Universal Robots PolyScope program: bearing_plate_pick.urp

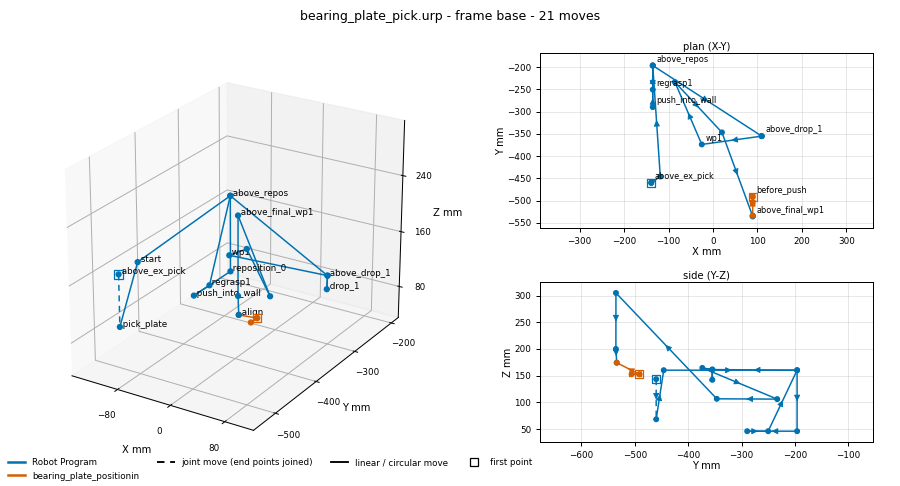
[picture p0: tool path of bearing_plate_pick.urp in frame base, 21 of 22 moves have a stored position in this frame; points joined in program order, loops and branches not executed]
Program bearing_plate_pick (installation=default directory=/programs/wrs2020 createdIn=5.6.0.90886 lastSavedIn=5.9.1.1031110 robotSerialNumber=20205500180)
Calibrated DH parameters: a=[0, -0.425, -0.3922, 0, 0, 0]; d=[0.1625, 0, 0, 0.1333, 0.0997, 0.0996]; alpha=[1.570796, 0, 0, 1.570796, -1.570796, 0]; deltaTheta=[0, 0, 0, 0, 0, 0]
Robot Program (runOnlyOnce=true)
  MoveJ speed 60 deg/s, acceleration 80 deg/s^2 (useActiveTCP=true) feature=Base
    currentpose := get_actual_tcp_pose()get_actual_joint_positions()
    Waypoint Waypoint (Variable): variable=currentpose
  MoveJ speed 60 deg/s, acceleration 80 deg/s^2 (useActiveTCP=true) feature=Base
    URCap Gripper (Robotiq_Grippers, Robotiq Inc.) dataModel(position=64.70588235294117, force=0.0, speed=0.0, positionInDouble=64.70588235294117, forceInDouble=0.0, speedInDouble=0.0, slaveIds=[9], blocking=true)
    Waypoint above_ex_pick: TCP in base x=-139.039 y=-460.061 z=143.501 mm, rx=-2.2048 ry=-2.2054 rz=0.0296 rad; joints [58.139, -91.524, 110.219, -109.456, -91.532, 58.113] deg; TCP offset x=0 y=0 z=220 mm, rx=0 ry=0 rz=0 rad
    Waypoint pick_plate: TCP in base x=-139.031 y=-460.052 z=68.363 mm, rx=-2.2048 ry=-2.2054 rz=0.0296 rad; joints [58.14, -86.891, 117.616, -121.485, -91.533, 58.114] deg; TCP offset x=0 y=0 z=220 mm, rx=0 ry=0 rz=0 rad
    URCap Gripper (Robotiq_Grippers, Robotiq Inc.) dataModel(position=100.0, force=0.0, speed=0.0, positionInDouble=100.0, forceInDouble=0.0, speedInDouble=0.0, slaveIds=[9], blocking=true)
  Folder Rearrange
    MoveL speed 800 mm/s, acceleration 1200 mm/s^2 (useActiveTCP=false) tcp=gripper_140_tip; feature=Base
      Waypoint start: motionParameters(blendRadius=0.03); TCP in base x=-118.669 y=-445.946 z=160.266 mm, rx=2.1923 ry=2.2501 rz=0.0089 rad; joints [58.256, -94.58, 110.219, -105.321, -89.927, 56.766] deg; TCP offset x=0 y=0 z=220 mm, rx=0 ry=0 rz=0 rad
      Waypoint above_repos: motionParameters(blendRadius=0.05); TCP in base x=-135.607 y=-196.202 z=160.258 mm, rx=3.137 ry=-0.0475 rz=0.0061 rad; joints [20.876, -133.857, 132.235, -88.26, -89.695, 112.61] deg; TCP offset x=0 y=0 z=220 mm, rx=0 ry=0 rz=0 rad
      Waypoint reposition_0: TCP in base x=-135.6 y=-196.2 z=46.036 mm, rx=3.1371 ry=-0.0475 rz=0.0061 rad; joints [20.876, -130.464, 148.282, -107.699, -89.695, 112.611] deg
      URCap Gripper (Robotiq_Grippers, Robotiq Inc.) dataModel(position=72.54901960784314, force=0.0, speed=0.0, positionInDouble=72.54901960784314, forceInDouble=0.0, speedInDouble=0.0, slaveIds=[9], blocking=true)
      URCap Gripper (Robotiq_Grippers, Robotiq Inc.) dataModel(position=83.92156862745098, force=0.0, speed=0.0, positionInDouble=83.92156862745098, forceInDouble=0.0, speedInDouble=0.0, slaveIds=[9], blocking=true)
      Waypoint push_into_wall: TCP in base x=-135.617 y=-289.652 z=46.047 mm, rx=3.137 ry=-0.0475 rz=0.0061 rad; joints [39.919, -110.73, 140.431, -119.691, -89.673, 131.655] deg
      URCap Gripper (Robotiq_Grippers, Robotiq Inc.) dataModel(position=72.54901960784314, force=0.0, speed=0.0, positionInDouble=72.54901960784314, forceInDouble=0.0, speedInDouble=0.0, slaveIds=[9], blocking=true)
      Waypoint regrasp1: TCP in base x=-135.589 y=-250.402 z=46.038 mm, rx=3.1371 ry=-0.0475 rz=0.0061 rad; joints [33.242, -118.348, 144.167, -115.768, -89.677, 124.976] deg
      URCap Gripper (Robotiq_Grippers, Robotiq Inc.) dataModel(position=100.0, force=0.0, speed=0.0, positionInDouble=100.0, forceInDouble=0.0, speedInDouble=0.0, slaveIds=[9], blocking=true)
      Waypoint above_repos: TCP in base x=-135.607 y=-196.202 z=160.258 mm, rx=3.137 ry=-0.0475 rz=0.0061 rad; joints [20.876, -133.857, 132.235, -88.26, -89.695, 112.61] deg
      URCap Gripper (Robotiq_Grippers, Robotiq Inc.) dataModel(position=100.0, force=0.0, speed=0.0, positionInDouble=100.0, forceInDouble=0.0, speedInDouble=0.0, slaveIds=[9], blocking=true)
  MoveL speed 800 mm/s, acceleration 1200 mm/s^2 (useActiveTCP=false) tcp=gripper_140_tip; feature=Base
    SuppressedNode
      Waypoint start: TCP in base x=-118.669 y=-445.946 z=160.266 mm, rx=2.1923 ry=2.2501 rz=0.0089 rad; joints [58.256, -94.58, 110.219, -105.321, -89.927, 56.766] deg; TCP offset x=0 y=0 z=220 mm, rx=0 ry=0 rz=0 rad
    Waypoint above_drop_1: TCP in base x=109.642 y=-355.035 z=161.42 mm, rx=0.0416 ry=-3.1373 rz=-0.0063 rad; joints [86.366, -108.401, 120.826, -102.213, -90.247, -5.154] deg; TCP offset x=0 y=0 z=220 mm, rx=0 ry=0 rz=0 rad
    Waypoint drop_1: TCP in base x=109 y=-355.041 z=142.278 mm, rx=0.0417 ry=-3.1373 rz=-0.0063 rad; joints [86.261, -107.694, 123.246, -105.338, -90.248, -5.26] deg; TCP offset x=0 y=0 z=220 mm, rx=0 ry=0 rz=0 rad
    URCap Gripper (Robotiq_Grippers, Robotiq Inc.) dataModel(position=72.54901960784314, force=0.0, speed=0.0, positionInDouble=72.54901960784314, forceInDouble=0.0, speedInDouble=0.0, slaveIds=[9], blocking=true)
    Waypoint above_drop_1: TCP in base x=109.642 y=-355.035 z=161.42 mm, rx=0.0416 ry=-3.1373 rz=-0.0063 rad; joints [86.366, -108.401, 120.826, -102.213, -90.247, -5.154] deg; TCP offset x=0 y=0 z=220 mm, rx=0 ry=0 rz=0 rad
    Waypoint wp1: motionParameters(blendRadius=0.05); TCP in base x=-25.271 y=-373.698 z=164.531 mm, rx=0.4375 ry=2.7113 rz=-0.1186 rad; joints [44.743, -110.618, 123.094, -92.727, -69.038, -28.731] deg; TCP offset x=0 y=0 z=220 mm, rx=0 ry=0 rz=0 rad
    Waypoint before_grasp: motionParameters(jointSpeed=1.047198 jointAcceleration=1.396263 cartesianSpeed=0.25 cartesianAcceleration=1.2 blendRadius=0.02); TCP in base x=-85.778 y=-233.44 z=106.112 mm, rx=0.6196 ry=1.477 rz=-0.6265 rad; joints [-24.668, -72.215, 139.816, -67.364, -68.98, -90.257] deg
    Waypoint at_grasp: motionParameters(jointSpeed=1.047198 jointAcceleration=1.396263 cartesianSpeed=0.25 cartesianAcceleration=1.2); TCP in base x=20.032 y=-346.58 z=106.691 mm, rx=0.6197 ry=1.477 rz=-0.6265 rad; joints [-4.452, -79.298, 152.241, -72.65, -48.761, -90.363] deg
    URCap Gripper (Robotiq_Grippers, Robotiq Inc.) dataModel(position=100.0, force=0.0, speed=0.0, positionInDouble=100.0, forceInDouble=0.0, speedInDouble=0.0, slaveIds=[9], blocking=true)
    MoveDirectionNode (toolParams=0.8, 0.4) expression=[-0.3,0.0,1.0]
      Until DISTANCE (allowActions=false deceleration=3 distanceNodeType=BLEND) Distance=0.15; motionParameters(blendRadius=0.08)
    Waypoint above_final_wp1: motionParameters(jointSpeed=1.047198 jointAcceleration=1.396263 cartesianSpeed=0.8 cartesianAcceleration=0.4 blendRadius=0.03); TCP in base x=89.208 y=-535.392 z=304.9 mm, rx=0.0022 ry=-2.7904 rz=1.4282 rad; joints [80.944, -112.949, 134.272, -165.222, -82.979, -5.575] deg
    Waypoint place: motionParameters(jointSpeed=1.047198 jointAcceleration=1.396263 cartesianSpeed=0.8 cartesianAcceleration=0.4); TCP in base x=89.218 y=-535.49 z=200.099 mm, rx=0.0021 ry=-2.8448 rz=1.3158 rad; joints [81.498, -103.024, 141.717, -178.058, -83.875, -5.768] deg
    URCap Gripper (Robotiq_Grippers, Robotiq Inc.) dataModel(position=72.54901960784314, force=0.0, speed=0.0, positionInDouble=72.54901960784314, forceInDouble=0.0, speedInDouble=0.0, slaveIds=[9], blocking=true)
    Waypoint align: TCP in base x=89.24 y=-533.942 z=174.306 mm, rx=0.0138 ry=2.8434 rz=-1.3083 rad; joints [80.63, -99.836, 144.208, -183.367, -82.506, -5.396] deg
    URCap Gripper (Robotiq_Grippers, Robotiq Inc.) dataModel(position=100.0, force=0.0, speed=0.0, positionInDouble=100.0, forceInDouble=0.0, speedInDouble=0.0, slaveIds=[9], blocking=true)
    URCap Gripper (Robotiq_Grippers, Robotiq Inc.) dataModel(position=72.54901960784314, force=0.0, speed=0.0, positionInDouble=72.54901960784314, forceInDouble=0.0, speedInDouble=0.0, slaveIds=[9], blocking=true)
  Call bearing_plate_positioning
SubProgram -> bearing_plate_positioning
SubProgram bearing_plate_positioning (keepSynchronizedWithDisk=true) programFile=/programs/wrs2020/bearing_plate_positioning.urp
  MoveL speed 250 mm/s, acceleration 1200 mm/s^2 (useActiveTCP=false) tcp=gripper_140_tip; feature=Base
    Waypoint before_push: TCP in base x=89.187 y=-491.509 z=152.605 mm, rx=0.003 ry=-2.9506 rz=1.0578 rad; joints [81.384, -106.52, 143.063, -165.713, -84.882, -6.911] deg
  URCap Gripper (Robotiq_Grippers, Robotiq Inc.) dataModel(position=100.0, force=0.0, speed=0.0, positionInDouble=100.0, forceInDouble=0.0, speedInDouble=0.0, slaveIds=[9], blocking=true)
  MoveL speed 250 mm/s, acceleration 1200 mm/s^2 (useActiveTCP=false) tcp=gripper_140_tip; feature=Base
    Waypoint push_end: motionParameters(jointSpeed=1.047198 jointAcceleration=1.396263 cartesianSpeed=0.05 cartesianAcceleration=0.02); TCP in base x=89.184 y=-506.034 z=152.639 mm, rx=0.003 ry=-2.9506 rz=1.0579 rad; joints [81.819, -103.812, 141.322, -166.712, -85.157, -6.571] deg
    Waypoint before_push: motionParameters(jointSpeed=1.047198 jointAcceleration=1.396263 cartesianSpeed=0.25 cartesianAcceleration=0.5); TCP in base x=89.187 y=-491.509 z=152.605 mm, rx=0.003 ry=-2.9506 rz=1.0578 rad; joints [81.384, -106.52, 143.063, -165.713, -84.882, -6.911] deg
  URCap Gripper (Robotiq_Grippers, Robotiq Inc.) dataModel(position=51.76470588235294, force=100.0, speed=100.0, positionInDouble=51.76470588235294, forceInDouble=100.0, speedInDouble=100.0, slaveIds=[9], blocking=true)
  MoveL speed 500 mm/s, acceleration 800 mm/s^2 (useActiveTCP=false) tcp=gripper_140_tip; feature=Base
    SuppressedNode
      Waypoint Waypoint_2: TCP in base x=89.229 y=-495.285 z=194.846 mm, rx=0.0168 ry=3.034 rz=-0.7765 rad; joints [82.081, -107.449, 128.407, -139.394, -85.816, -6.224] deg
    Waypoint final_grasp: TCP in base x=89.247 y=-533.927 z=174.318 mm, rx=0.0137 ry=2.8434 rz=-1.3083 rad; joints [80.631, -99.839, 144.21, -183.366, -82.507, -5.398] deg
  URCap Gripper (Robotiq_Grippers, Robotiq Inc.) dataModel(position=100.0, force=0.0, speed=0.0, positionInDouble=100.0, forceInDouble=0.0, speedInDouble=0.0, slaveIds=[9], blocking=true)
  URCap Gripper (Robotiq_Grippers, Robotiq Inc.) dataModel(position=82.3529411764706, force=100.0, speed=0.0, positionInDouble=82.3529411764706, forceInDouble=100.0, speedInDouble=0.0, slaveIds=[9], blocking=true)
